TYPE E_FIO_PNP_State :
(
    Idle,
    MoveToPick,
    Grab,
    LiftAfterPick,
    MoveToPlace,
    Release,
    RetractAfterPlace,
    Error
);
END_TYPE

(* stored: Version 1.1.0.1
   DUT E_FIO_PNP_State: Id {07718223-ff70-4067-8f23-077aab32ef74} *)
